// Mitsubishi GX Developer project: пресс 70 отключение при простое   PLC: Q04UDEH

PROGRAM MAIN
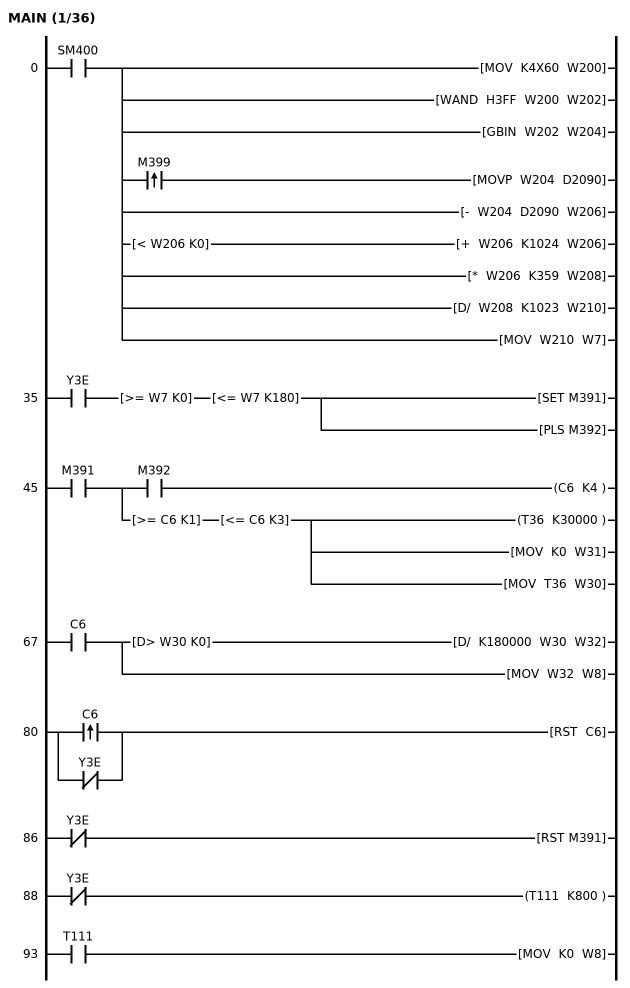
0     LD      SM400
      MOV     K4X60 W200
      WAND    H3FF W200 W202
      GBIN    W202 W204
      MPS
      ANDP    M399
      MOVP    W204 D2090
      MPP
      -       W204 D2090 W206
      MPS
      AND<    W206 K0
      +       W206 K1024 W206
      MPP
      *       W206 K359 W208
      D/      W208 K1023 W210
      MOV     W210 W7
35    LD      Y3E
      AND>=   W7 K0
      AND<=   W7 K180
      SET     M391
      PLS     M392
45    LD      M391
      MPS
      AND     M392
      OUT     C6 K4
      MPP
      AND>=   C6 K1
      AND<=   C6 K3
      OUTH    T36 K30000
      MOV     K0 W31
      MOV     T36 W30
67    LD      C6
      MPS
      ANDD>   W30 K0
      D/      K180000 W30 W32
      MPP
      MOV     W32 W8
80    LDP     C6
      ORI     Y3E
      RST     C6
86    LDI     Y3E
      RST     M391
88    LDI     Y3E
      OUT     T111 K800
93    LD      T111
      MOV     K0 W8
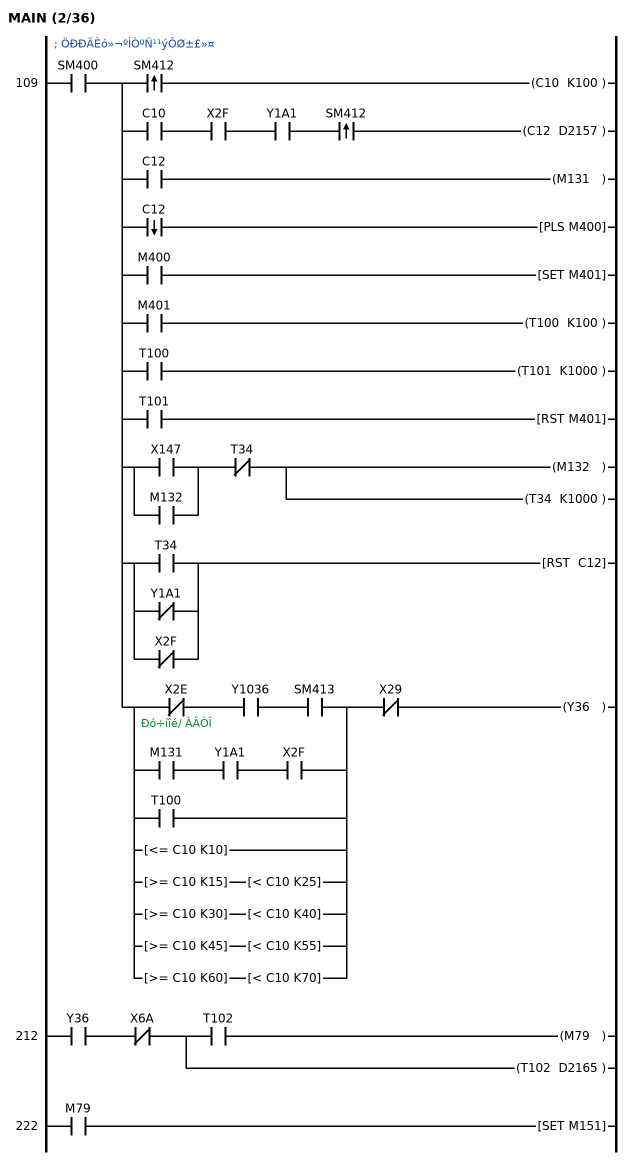
; 中心润滑和液压过载保护
109   LD      SM400
      MPS
      ANDP    SM412
      OUT     C10 K100
      MRD
      AND     C10
      AND     X2F
      AND     Y1A1
      ANDP    SM412
      OUT     C12 D2157
      MRD
      AND     C12
      OUT     M131
      MRD
      ANDF    C12
      PLS     M400
      MRD
      AND     M400
      SET     M401
      MRD
      AND     M401
      OUT     T100 K100
      MRD
      AND     T100
      OUT     T101 K1000
      MRD
      AND     T101
      RST     M401
      MRD
      LD      X147
      OR      M132
      ANB
      ANI     T34
      OUT     M132
      OUT     T34 K1000
      MRD
      LD      T34
      ORI     Y1A1
      ORI     X2F
      ANB
      RST     C12
      MPP
      LDI     X2E  ; Ручной/ АВТО
      AND     Y1036
      AND     SM413
      LD      M131
      AND     Y1A1
      AND     X2F
      ORB
      OR      T100
      OR<=    C10 K10
      LD>=    C10 K15
      AND<    C10 K25
      ORB
      LD>=    C10 K30
      AND<    C10 K40
      ORB
      LD>=    C10 K45
      AND<    C10 K55
      ORB
      LD>=    C10 K60
      AND<    C10 K70
      ORB
      ANB
      ANI     X29
      OUT     Y36
212   LD      Y36
      ANI     X6A
      MPS
      AND     T102
      OUT     M79
      MPP
      OUT     T102 D2165
222   LD      M79
      SET     M151
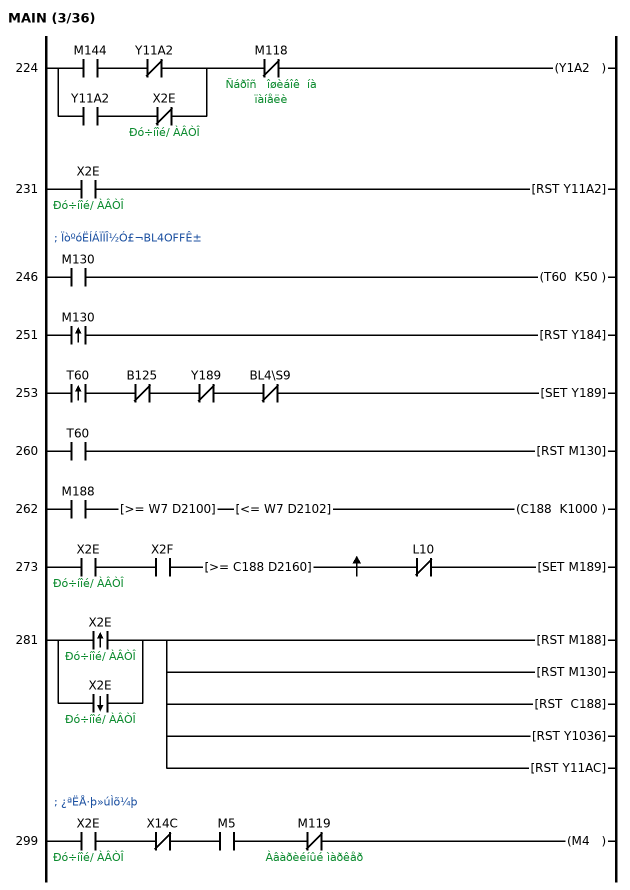
224   LD      M144
      ANI     Y11A2
      LD      Y11A2
      ANI     X2E  ; Ручной/ АВТО
      ORB
      ANI     M118  ; Сброс   ошибок  на панели
      OUT     Y1A2
231   LD      X2E  ; Ручной/ АВТО
      RST     Y11A2
; 向后送料衔接，BL4OFF时
246   LD      M130
      OUT     T60 K50
251   LDP     M130
      RST     Y184
253   LDP     T60
      ANI     B125
      ANI     Y189
      ANI     BL4\S9
      SET     Y189
260   LD      T60
      RST     M130
262   LD      M188
      AND>=   W7 D2100
      AND<=   W7 D2102
      OUT     C188 K1000
273   LD      X2E  ; Ручной/ АВТО
      AND     X2F
      AND>=   C188 D2160
      MEP
      ANI     L10
      SET     M189
281   LDP     X2E  ; Ручной/ АВТО
      ORF     X2E  ; Ручной/ АВТО
      RST     M188
      RST     M130
      RST     C188
      RST     Y1036
      RST     Y11AC
; 开伺服机条件
299   LD      X2E  ; Ручной/ АВТО
      ANI     X14C
      AND     M5
      ANI     M119  ; Аварийный маркер
      OUT     M4
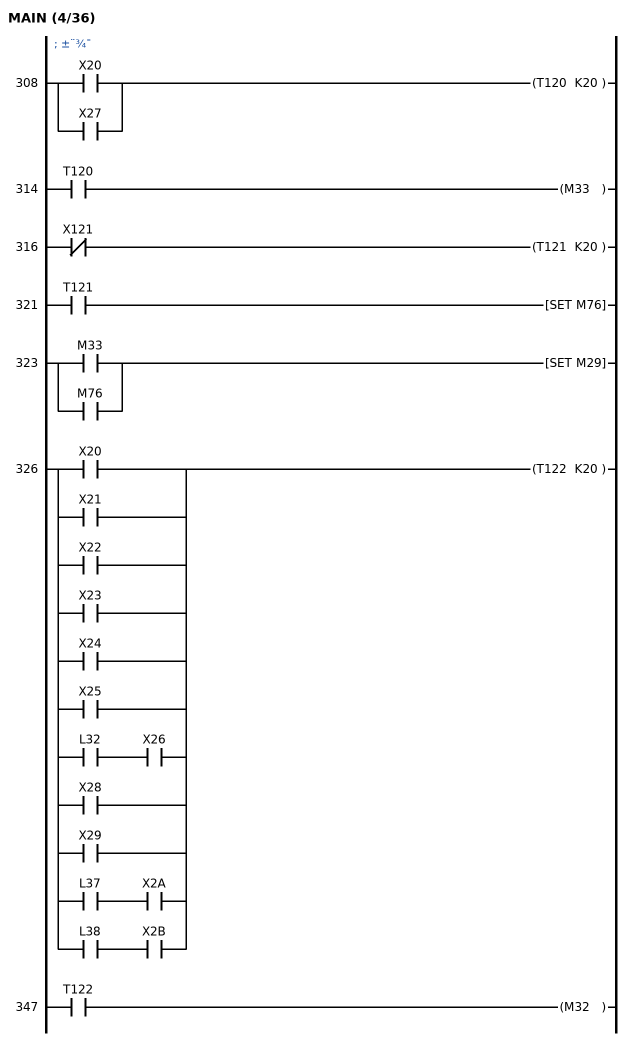
; ±¨¾¯
308   LD      X20
      OR      X27
      OUT     T120 K20
314   LD      T120
      OUT     M33
316   LDI     X121
      OUT     T121 K20
321   LD      T121
      SET     M76
323   LD      M33
      OR      M76
      SET     M29
326   LD      X20
      OR      X21
      OR      X22
      OR      X23
      OR      X24
      OR      X25
      LD      L32
      AND     X26
      ORB
      OR      X28
      OR      X29
      LD      L37
      AND     X2A
      ORB
      LD      L38
      AND     X2B
      ORB
      OUT     T122 K20
347   LD      T122
      OUT     M32
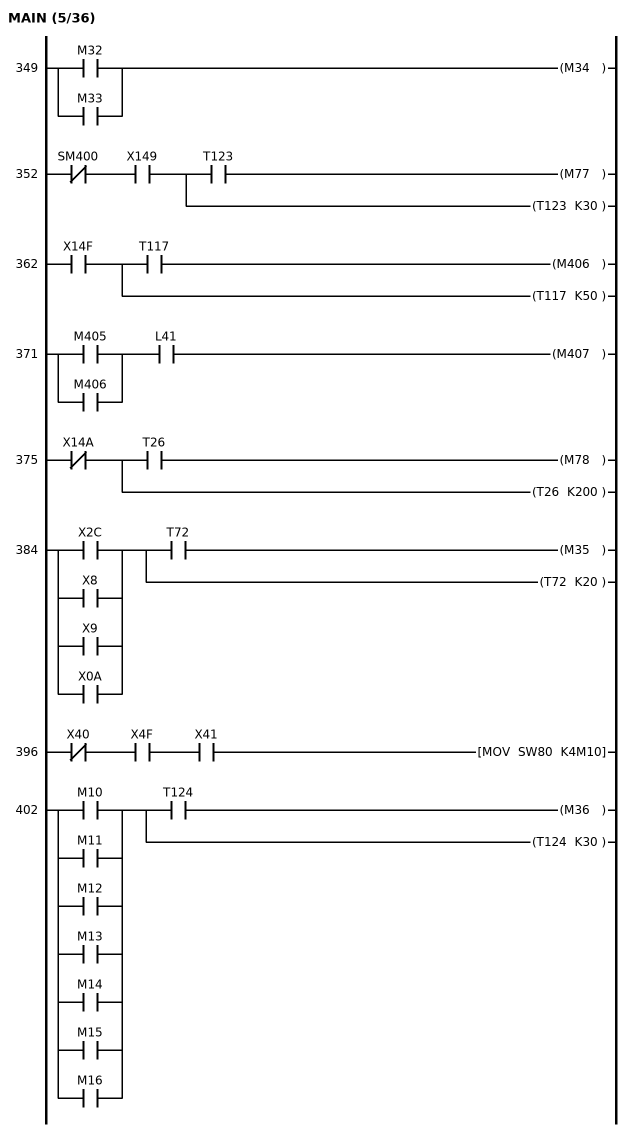
349   LD      M32
      OR      M33
      OUT     M34
352   LDI     SM400
      AND     X149
      MPS
      AND     T123
      OUT     M77
      MPP
      OUT     T123 K30
362   LD      X14F
      MPS
      AND     T117
      OUT     M406
      MPP
      OUT     T117 K50
371   LD      M405
      OR      M406
      AND     L41
      OUT     M407
375   LDI     X14A
      MPS
      AND     T26
      OUT     M78
      MPP
      OUT     T26 K200
384   LD      X2C
      OR      X8
      OR      X9
      OR      X0A
      MPS
      AND     T72
      OUT     M35
      MPP
      OUT     T72 K20
396   LDI     X40
      AND     X4F
      AND     X41
      MOV     SW80 K4M10
402   LD      M10
      OR      M11
      OR      M12
      OR      M13
      OR      M14
      OR      M15
      OR      M16
      MPS
      AND     T124
      OUT     M36
      MPP
      OUT     T124 K30
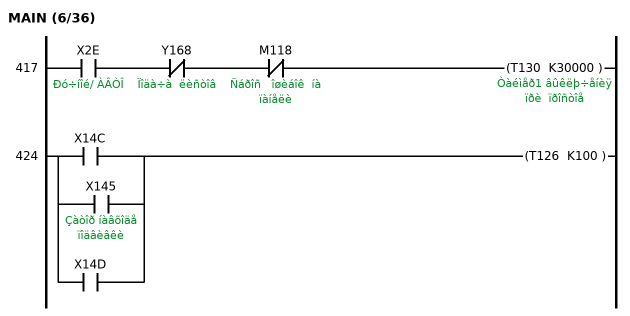
417   LD      X2E  ; Ручной/ АВТО
      ANI     Y168  ; Подача  листов
      ANI     M118  ; Сброс   ошибок  на панели
      OUT     T130 K30000  ; Таймер1 выключения при  простое
424   LD      X14C
      OR      X145  ; Затор навходе   подвивки
      OR      X14D
      OUTH    T126 K100
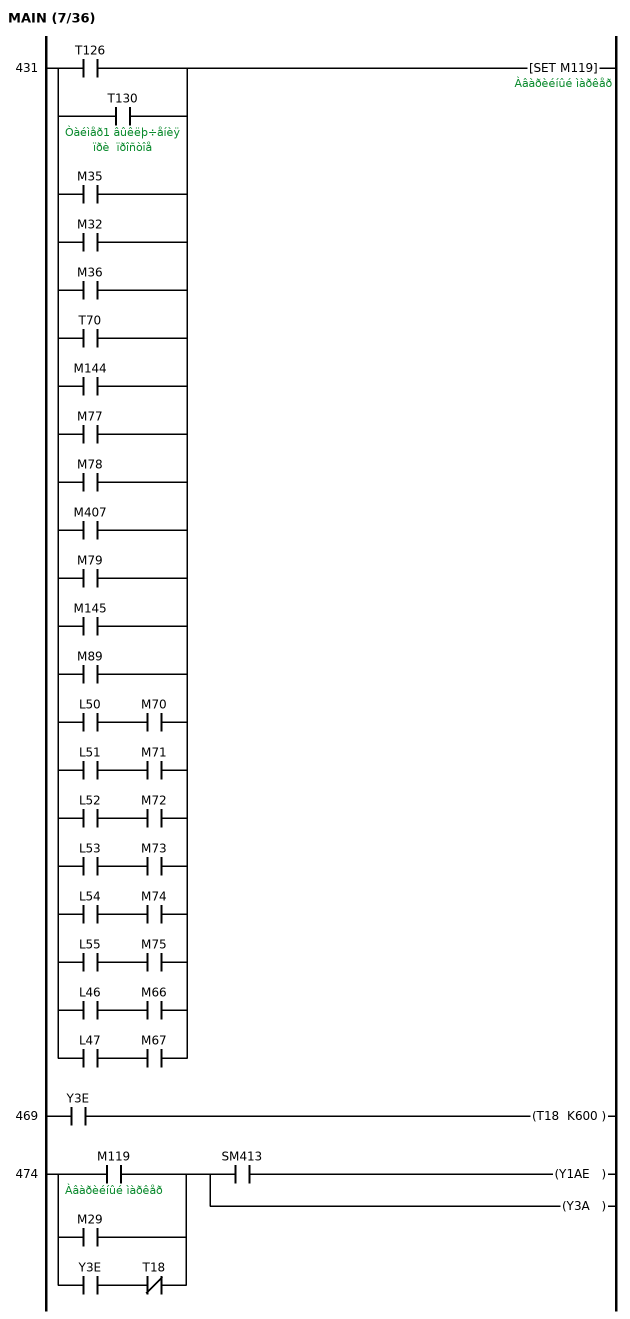
431   LD      T126
      OR      T130  ; Таймер1 выключения при  простое
      OR      M35
      OR      M32
      OR      M36
      OR      T70
      OR      M144
      OR      M77
      OR      M78
      OR      M407
      OR      M79
      OR      M145
      OR      M89
      LD      L50
      AND     M70
      ORB
      LD      L51
      AND     M71
      ORB
      LD      L52
      AND     M72
      ORB
      LD      L53
      AND     M73
      ORB
      LD      L54
      AND     M74
      ORB
      LD      L55
      AND     M75
      ORB
      LD      L46
      AND     M66
      ORB
      LD      L47
      AND     M67
      ORB
      SET     M119  ; Аварийный маркер
469   LD      Y3E
      OUT     T18 K600
474   LD      M119  ; Аварийный маркер
      OR      M29
      LD      Y3E
      ANI     T18
      ORB
      MPS
      AND     SM413
      OUT     Y1AE
      MPP
      OUT     Y3A
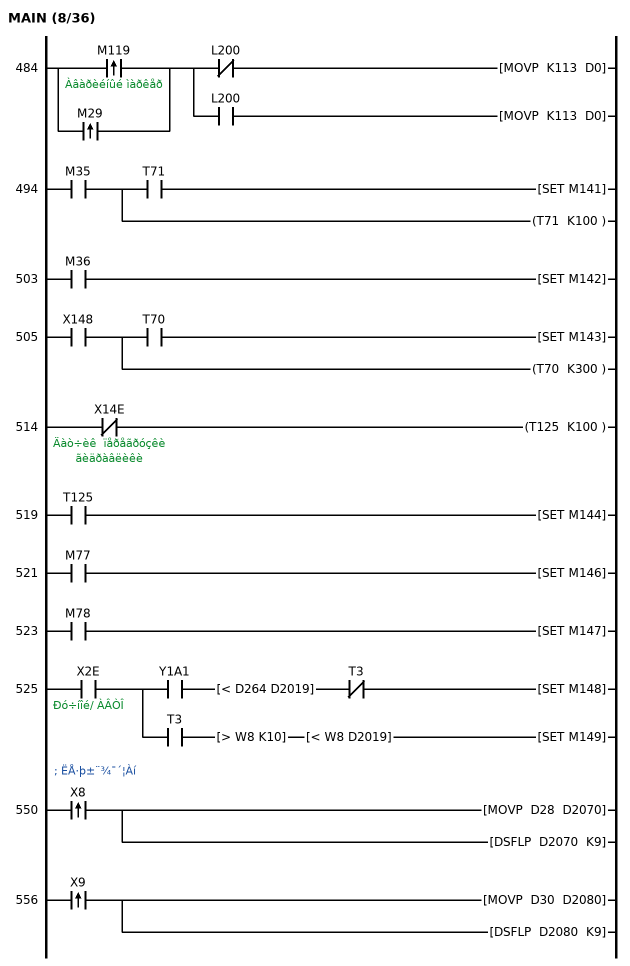
484   LDP     M119  ; Аварийный маркер
      ORP     M29
      MPS
      ANI     L200
      MOVP    K113 D0
      MPP
      AND     L200
      MOVP    K113 D0
494   LD      M35
      MPS
      AND     T71
      SET     M141
      MPP
      OUT     T71 K100
503   LD      M36
      SET     M142
505   LD      X148
      MPS
      AND     T70
      SET     M143
      MPP
      OUT     T70 K300
514   LDI     X14E  ; Датчик  перегрузки гидравлики
      OUTH    T125 K100
519   LD      T125
      SET     M144
521   LD      M77
      SET     M146
523   LD      M78
      SET     M147
525   LD      X2E  ; Ручной/ АВТО
      MPS
      AND     Y1A1
      AND<    D264 D2019
      ANI     T3
      SET     M148
      MPP
      AND     T3
      AND>    W8 K10
      AND<    W8 D2019
      SET     M149
; 伺服报警处理
550   LDP     X8
      MOVP    D28 D2070
      DSFLP   D2070 K9
556   LDP     X9
      MOVP    D30 D2080
      DSFLP   D2080 K9
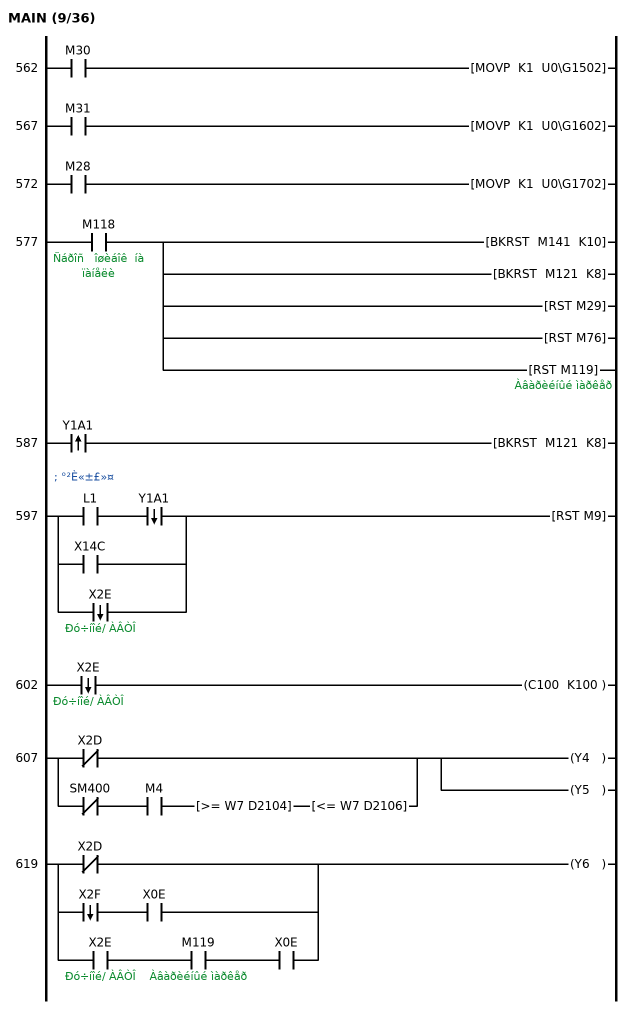
562   LD      M30
      MOVP    K1 U0\G1502
567   LD      M31
      MOVP    K1 U0\G1602
572   LD      M28
      MOVP    K1 U0\G1702
577   LD      M118  ; Сброс   ошибок  на панели
      BKRST   M141 K10
      BKRST   M121 K8
      RST     M29
      RST     M76
      RST     M119  ; Аварийный маркер
587   LDP     Y1A1
      BKRST   M121 K8
; 安全保护
597   LD      L1
      ANDF    Y1A1
      OR      X14C
      ORF     X2E  ; Ручной/ АВТО
      RST     M9
602   LDF     X2E  ; Ручной/ АВТО
      OUT     C100 K100
607   LDI     X2D
      LDI     SM400
      AND     M4
      AND>=   W7 D2104
      AND<=   W7 D2106
      ORB
      OUT     Y4
      OUT     Y5
619   LDI     X2D
      LDF     X2F
      AND     X0E
      ORB
      LD      X2E  ; Ручной/ АВТО
      AND     M119  ; Аварийный маркер
      AND     X0E
      ORB
      OUT     Y6
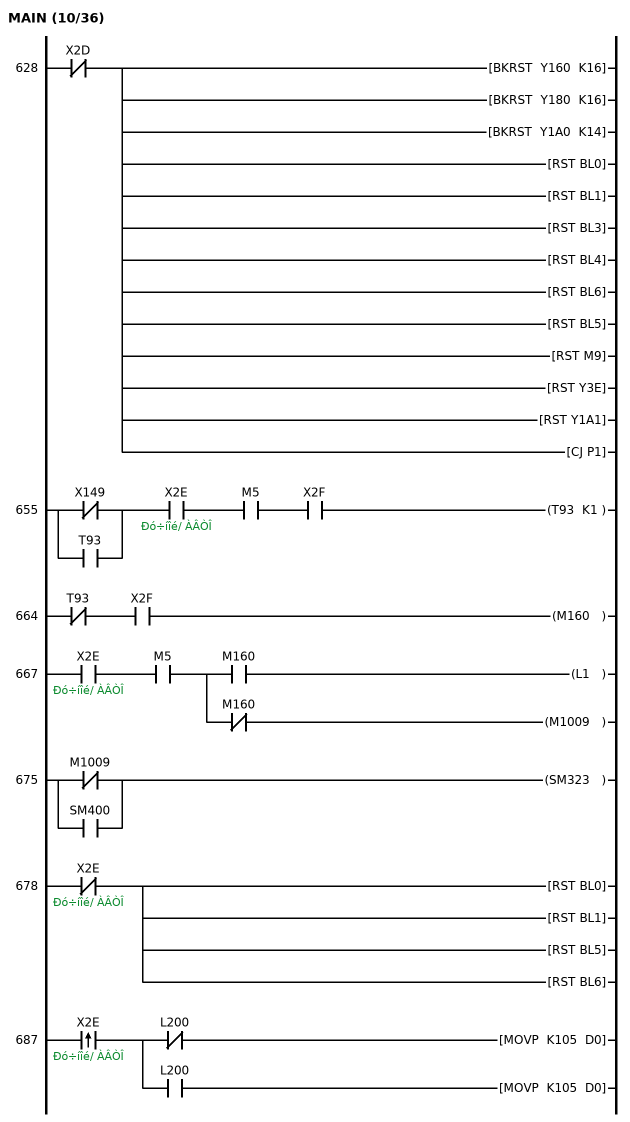
628   LDI     X2D
      BKRST   Y160 K16
      BKRST   Y180 K16
      BKRST   Y1A0 K14
      RST     BL0
      RST     BL1
      RST     BL3
      RST     BL4
      RST     BL6
      RST     BL5
      RST     M9
      RST     Y3E
      RST     Y1A1
      CJ      P1
655   LDI     X149
      OR      T93
      AND     X2E  ; Ручной/ АВТО
      AND     M5
      AND     X2F
      OUT     T93 K1
664   LDI     T93
      AND     X2F
      OUT     M160
667   LD      X2E  ; Ручной/ АВТО
      AND     M5
      MPS
      AND     M160
      OUT     L1
      MPP
      ANI     M160
      OUT     M1009
675   LDI     M1009
      OR      SM400
      OUT     SM323
678   LDI     X2E  ; Ручной/ АВТО
      RST     BL0
      RST     BL1
      RST     BL5
      RST     BL6
687   LDP     X2E  ; Ручной/ АВТО
      MPS
      ANI     L200
      MOVP    K105 D0
      MPP
      AND     L200
      MOVP    K105 D0
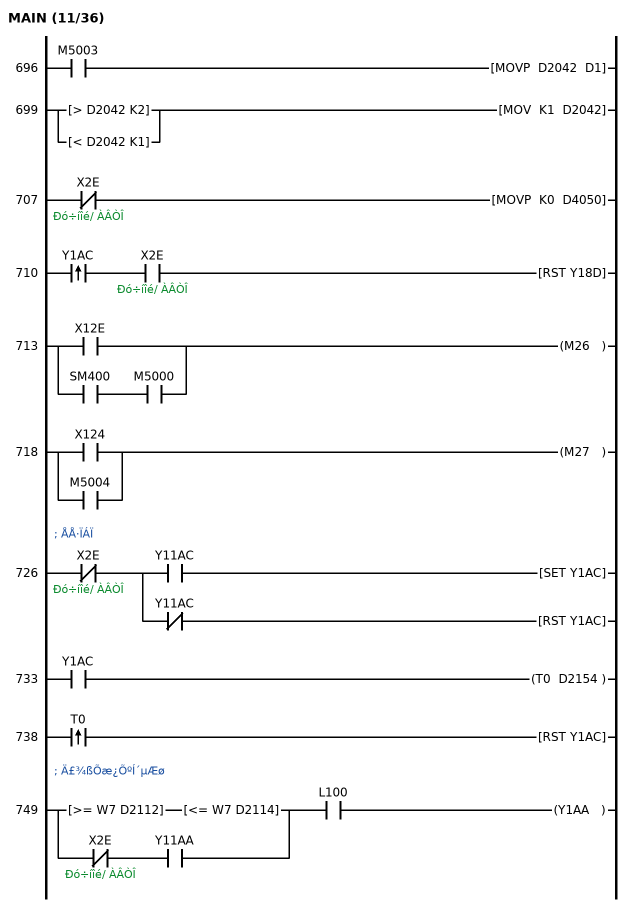
696   LD      M5003
      MOVP    D2042 D1
699   LD>     D2042 K2
      OR<     D2042 K1
      MOV     K1 D2042
707   LDI     X2E  ; Ручной/ АВТО
      MOVP    K0 D4050
710   LDP     Y1AC
      AND     X2E  ; Ручной/ АВТО
      RST     Y18D
713   LD      X12E
      LD      SM400
      AND     M5000
      ORB
      OUT     M26
718   LD      X124
      OR      M5004
      OUT     M27
; ÅÅ·ÏÁÏ
726   LDI     X2E  ; Ручной/ АВТО
      MPS
      AND     Y11AC
      SET     Y1AC
      MPP
      ANI     Y11AC
      RST     Y1AC
733   LD      Y1AC
      OUTH    T0 D2154
738   LDP     T0
      RST     Y1AC
; Ä£¾ßÕæ¿ÕºÍ´µÆø
749   LD>=    W7 D2112
      AND<=   W7 D2114
      LDI     X2E  ; Ручной/ АВТО
      AND     Y11AA
      ORB
      AND     L100
      OUT     Y1AA
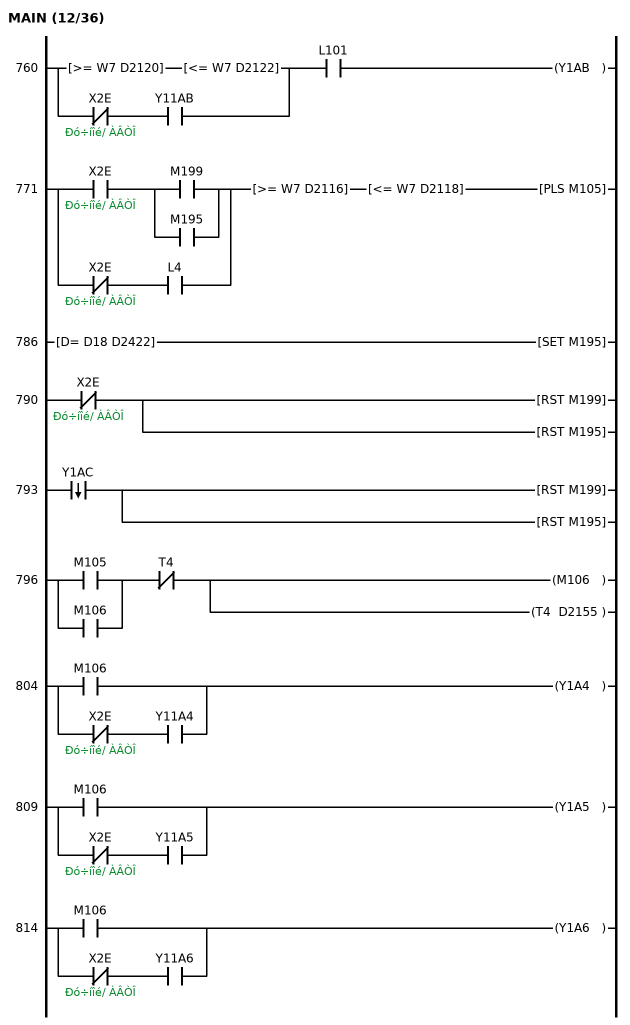
760   LD>=    W7 D2120
      AND<=   W7 D2122
      LDI     X2E  ; Ручной/ АВТО
      AND     Y11AB
      ORB
      AND     L101
      OUT     Y1AB
771   LD      X2E  ; Ручной/ АВТО
      LD      M199
      OR      M195
      ANB
      LDI     X2E  ; Ручной/ АВТО
      AND     L4
      ORB
      AND>=   W7 D2116
      AND<=   W7 D2118
      PLS     M105
786   LDD=    D18 D2422
      SET     M195
790   LDI     X2E  ; Ручной/ АВТО
      RST     M199
      RST     M195
793   LDF     Y1AC
      RST     M199
      RST     M195
796   LD      M105
      OR      M106
      ANI     T4
      OUT     M106
      OUTH    T4 D2155
804   LD      M106
      LDI     X2E  ; Ручной/ АВТО
      AND     Y11A4
      ORB
      OUT     Y1A4
809   LD      M106
      LDI     X2E  ; Ручной/ АВТО
      AND     Y11A5
      ORB
      OUT     Y1A5
814   LD      M106
      LDI     X2E  ; Ручной/ АВТО
      AND     Y11A6
      ORB
      OUT     Y1A6
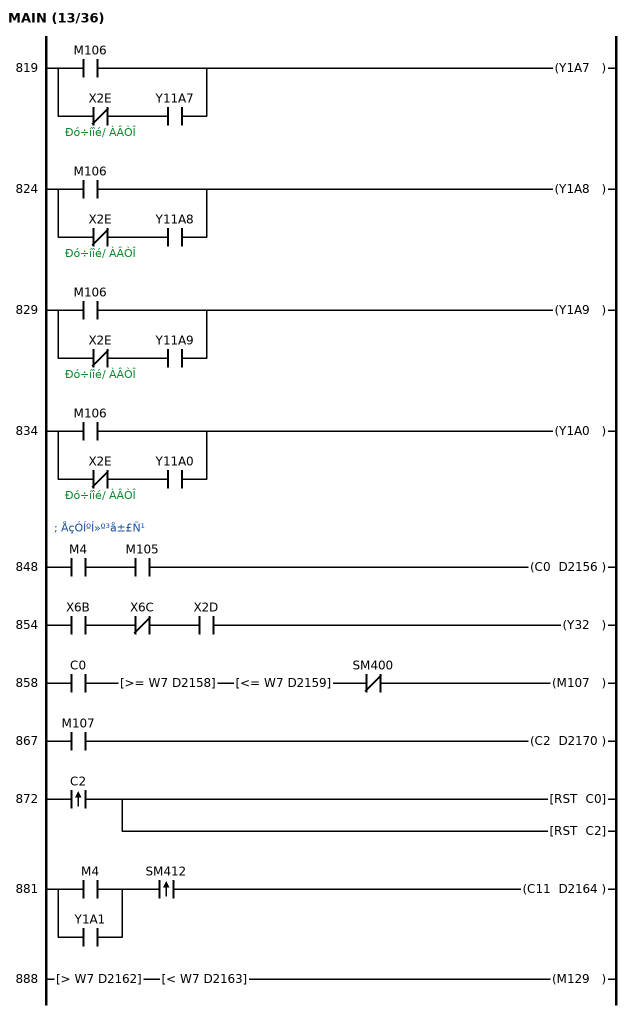
819   LD      M106
      LDI     X2E  ; Ручной/ АВТО
      AND     Y11A7
      ORB
      OUT     Y1A7
824   LD      M106
      LDI     X2E  ; Ручной/ АВТО
      AND     Y11A8
      ORB
      OUT     Y1A8
829   LD      M106
      LDI     X2E  ; Ручной/ АВТО
      AND     Y11A9
      ORB
      OUT     Y1A9
834   LD      M106
      LDI     X2E  ; Ручной/ АВТО
      AND     Y11A0
      ORB
      OUT     Y1A0
; ÅçÓÍºÍ»º³å±£Ñ¹
848   LD      M4
      AND     M105
      OUT     C0 D2156
854   LD      X6B
      ANI     X6C
      AND     X2D
      OUT     Y32
858   LD      C0
      AND>=   W7 D2158
      AND<=   W7 D2159
      ANI     SM400
      OUT     M107
867   LD      M107
      OUT     C2 D2170
872   LDP     C2
      RST     C0
      RST     C2
881   LD      M4
      OR      Y1A1
      ANDP    SM412
      OUT     C11 D2164
888   LD>     W7 D2162
      AND<    W7 D2163
      OUT     M129
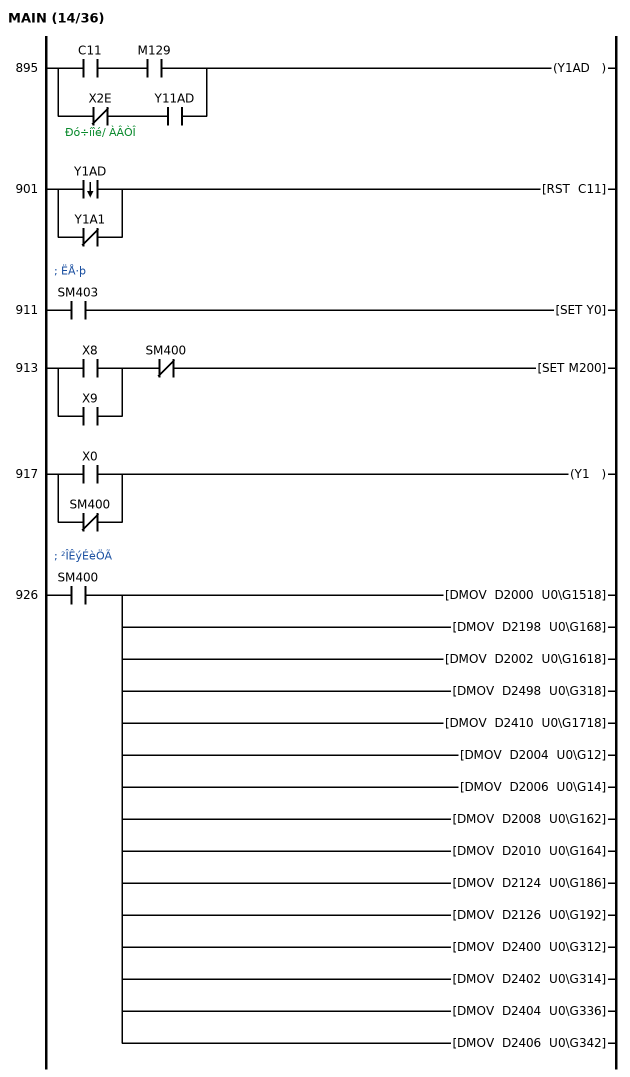
895   LD      C11
      AND     M129
      LDI     X2E  ; Ручной/ АВТО
      AND     Y11AD
      ORB
      OUT     Y1AD
901   LDF     Y1AD
      ORI     Y1A1
      RST     C11
; ËÅ·þ
911   LD      SM403
      SET     Y0
913   LD      X8
      OR      X9
      ANI     SM400
      SET     M200
917   LD      X0
      ORI     SM400
      OUT     Y1
; 参数设置
926   LD      SM400
      DMOV    D2000 U0\G1518
      DMOV    D2198 U0\G168
      DMOV    D2002 U0\G1618
      DMOV    D2498 U0\G318
      DMOV    D2410 U0\G1718
      DMOV    D2004 U0\G12
      DMOV    D2006 U0\G14
      DMOV    D2008 U0\G162
      DMOV    D2010 U0\G164
      DMOV    D2124 U0\G186
      DMOV    D2126 U0\G192
      DMOV    D2400 U0\G312
      DMOV    D2402 U0\G314
      DMOV    D2404 U0\G336
      DMOV    D2406 U0\G342
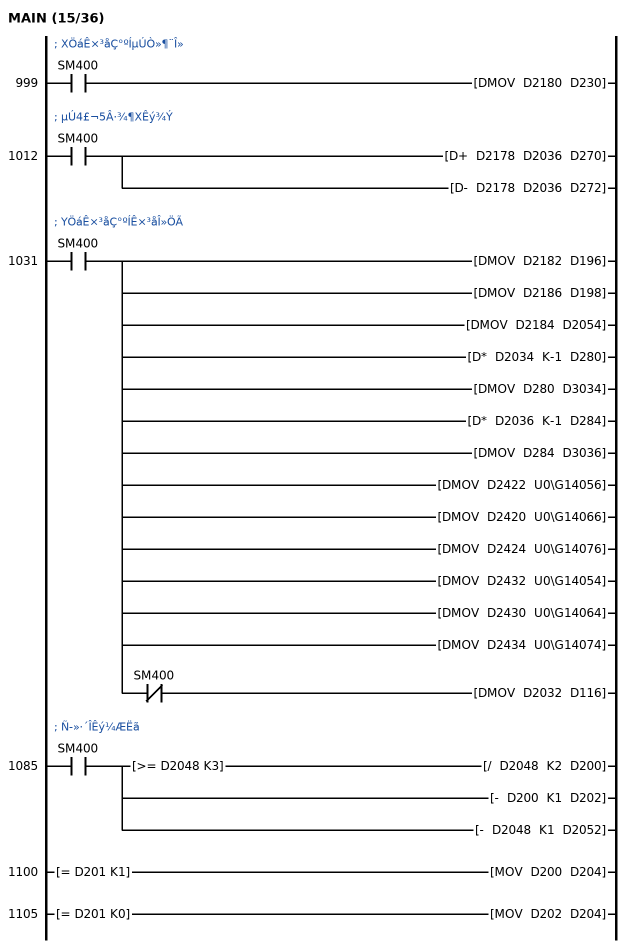
; X轴首冲前和第一定位
999   LD      SM400
      DMOV    D2180 D230
; 第4，5路径X数据
1012  LD      SM400
      D+      D2178 D2036 D270
      D-      D2178 D2036 D272
; Y轴首冲前和首冲位置
1031  LD      SM400
      DMOV    D2182 D196
      DMOV    D2186 D198
      DMOV    D2184 D2054
      D*      D2034 K-1 D280
      DMOV    D280 D3034
      D*      D2036 K-1 D284
      DMOV    D284 D3036
      DMOV    D2422 U0\G14056
      DMOV    D2420 U0\G14066
      DMOV    D2424 U0\G14076
      DMOV    D2432 U0\G14054
      DMOV    D2430 U0\G14064
      DMOV    D2434 U0\G14074
      ANI     SM400
      DMOV    D2032 D116
; 循环次数计算
1085  LD      SM400
      MPS
      AND>=   D2048 K3
      /       D2048 K2 D200
      MPP
      -       D200 K1 D202
      -       D2048 K1 D2052
1100  LD=     D201 K1
      MOV     D200 D204
1105  LD=     D201 K0
      MOV     D202 D204
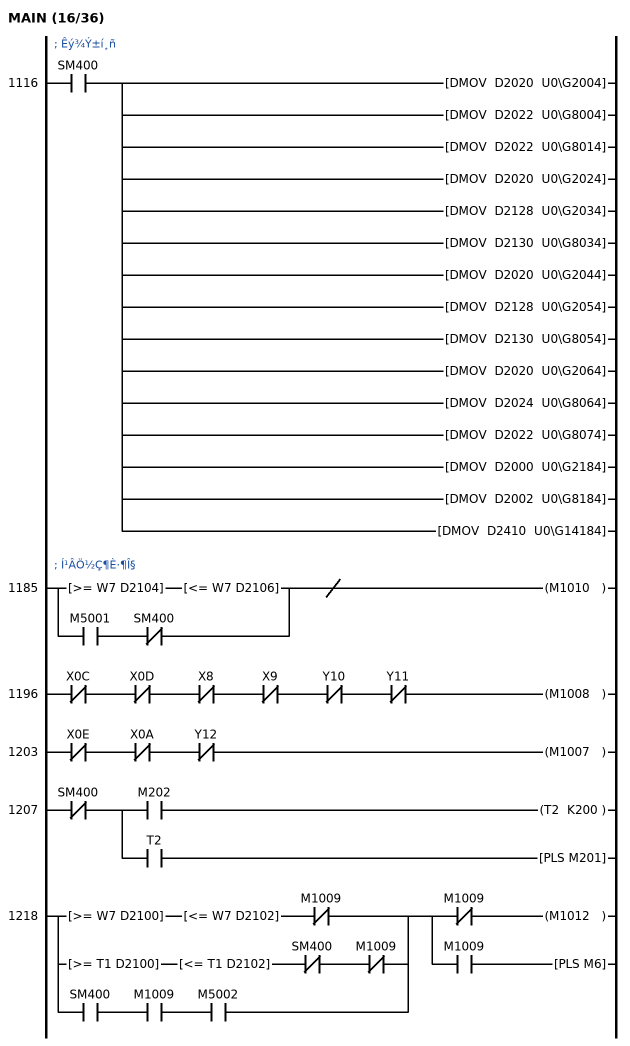
; 数据表格
1116  LD      SM400
      DMOV    D2020 U0\G2004
      DMOV    D2022 U0\G8004
      DMOV    D2022 U0\G8014
      DMOV    D2020 U0\G2024
      DMOV    D2128 U0\G2034
      DMOV    D2130 U0\G8034
      DMOV    D2020 U0\G2044
      DMOV    D2128 U0\G2054
      DMOV    D2130 U0\G8054
      DMOV    D2020 U0\G2064
      DMOV    D2024 U0\G8064
      DMOV    D2022 U0\G8074
      DMOV    D2000 U0\G2184
      DMOV    D2002 U0\G8184
      DMOV    D2410 U0\G14184
; 凸轮角度范围
1185  LD>=    W7 D2104
      AND<=   W7 D2106
      LD      M5001
      ANI     SM400
      ORB
      INV
      OUT     M1010
1196  LDI     X0C
      ANI     X0D
      ANI     X8
      ANI     X9
      ANI     Y10
      ANI     Y11
      OUT     M1008
1203  LDI     X0E
      ANI     X0A
      ANI     Y12
      OUT     M1007
1207  LDI     SM400
      MPS
      AND     M202
      OUT     T2 K200
      MPP
      AND     T2
      PLS     M201
1218  LD>=    W7 D2100
      AND<=   W7 D2102
      ANI     M1009
      LD>=    T1 D2100
      AND<=   T1 D2102
      ANI     SM400
      ANI     M1009
      ORB
      LD      SM400
      AND     M1009
      AND     M5002
      ORB
      MPS
      ANI     M1009
      OUT     M1012
      MPP
      AND     M1009
      PLS     M6
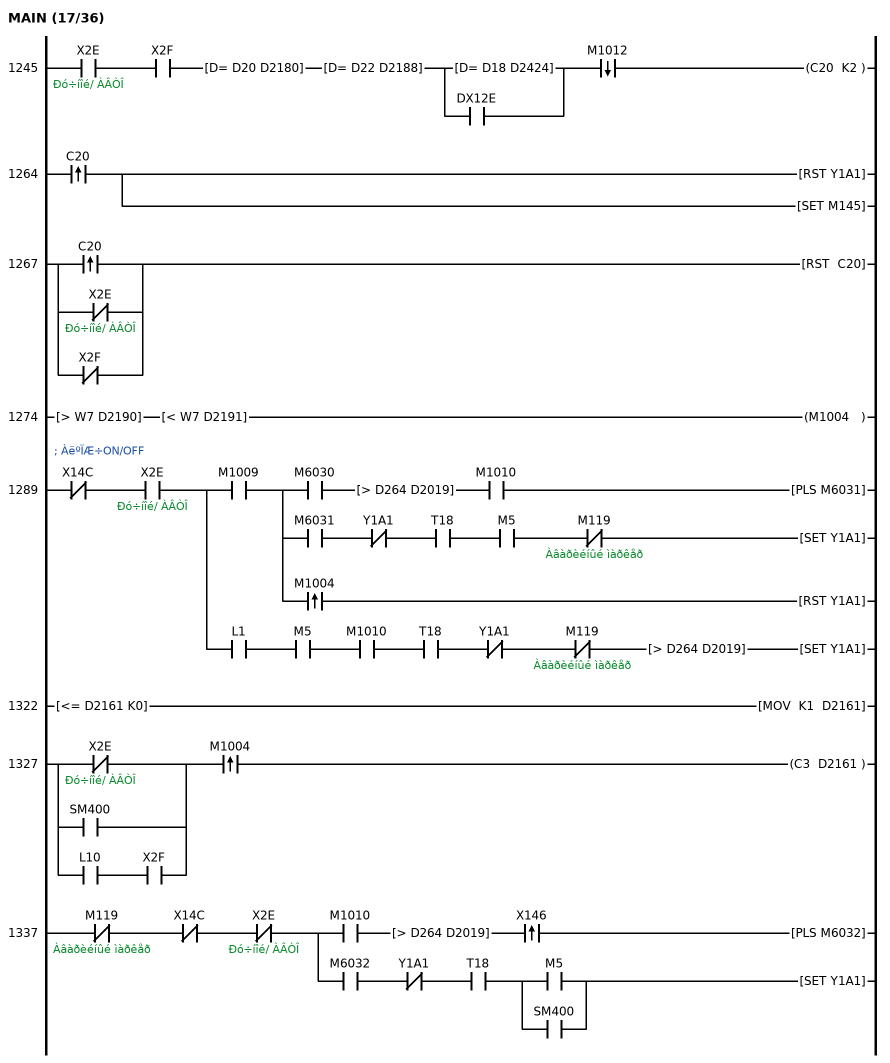
1245  LD      X2E  ; Ручной/ АВТО
      AND     X2F
      ANDD=   D20 D2180
      ANDD=   D22 D2188
      LDD=    D18 D2424
      OR      DX12E
      ANB
      ANDF    M1012
      OUT     C20 K2
1264  LDP     C20
      RST     Y1A1
      SET     M145
1267  LDP     C20
      ORI     X2E  ; Ручной/ АВТО
      ORI     X2F
      RST     C20
1274  LD>     W7 D2190
      AND<    W7 D2191
      OUT     M1004
; 离合器ON/OFF
1289  LDI     X14C
      AND     X2E  ; Ручной/ АВТО
      MPS
      AND     M1009
      MPS
      AND     M6030
      AND>    D264 D2019
      AND     M1010
      PLS     M6031
      MRD
      AND     M6031
      ANI     Y1A1
      AND     T18
      AND     M5
      ANI     M119  ; Аварийный маркер
      SET     Y1A1
      MPP
      ANDP    M1004
      RST     Y1A1
      MPP
      AND     L1
      AND     M5
      AND     M1010
      AND     T18
      ANI     Y1A1
      ANI     M119  ; Аварийный маркер
      AND>    D264 D2019
      SET     Y1A1
1322  LD<=    D2161 K0
      MOV     K1 D2161
1327  LDI     X2E  ; Ручной/ АВТО
      OR      SM400
      LD      L10
      AND     X2F
      ORB
      ANDP    M1004
      OUT     C3 D2161
1337  LDI     M119  ; Аварийный маркер
      ANI     X14C
      ANI     X2E  ; Ручной/ АВТО
      MPS
      AND     M1010
      AND>    D264 D2019
      ANDP    X146
      PLS     M6032
      MPP
      AND     M6032
      ANI     Y1A1
      AND     T18
      LD      M5
      OR      SM400
      ANB
      SET     Y1A1
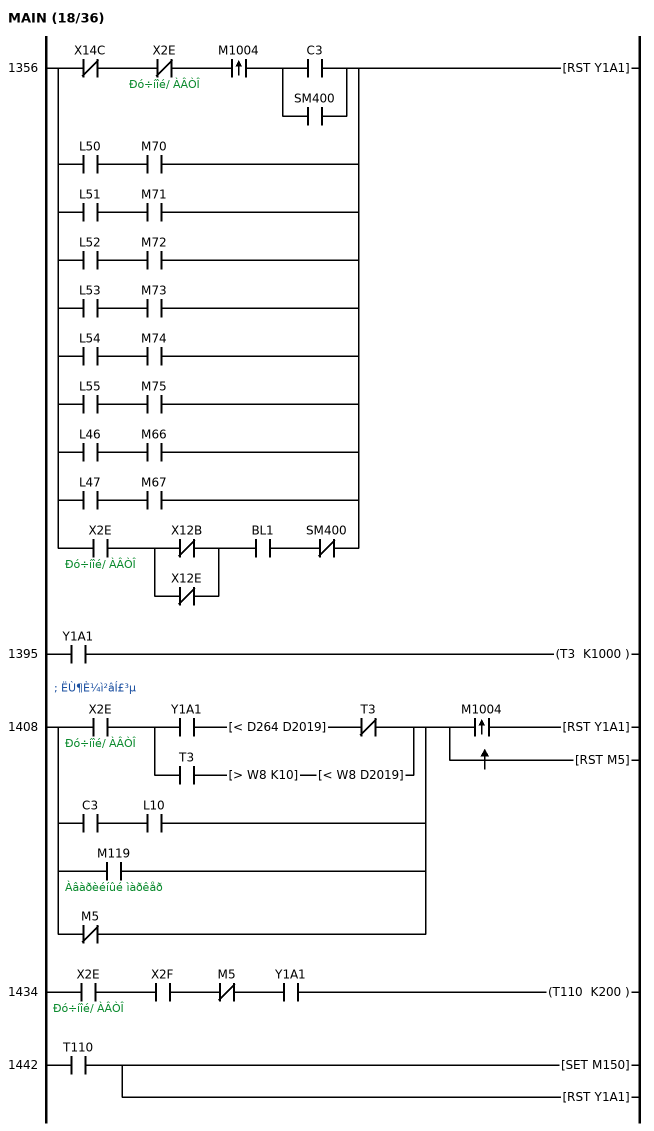
1356  LDI     X14C
      ANI     X2E  ; Ручной/ АВТО
      ANDP    M1004
      LD      C3
      OR      SM400
      ANB
      LD      L50
      AND     M70
      ORB
      LD      L51
      AND     M71
      ORB
      LD      L52
      AND     M72
      ORB
      LD      L53
      AND     M73
      ORB
      LD      L54
      AND     M74
      ORB
      LD      L55
      AND     M75
      ORB
      LD      L46
      AND     M66
      ORB
      LD      L47
      AND     M67
      ORB
      LD      X2E  ; Ручной/ АВТО
      LDI     X12B
      ORI     X12E
      ANB
      AND     BL1
      ANI     SM400
      ORB
      RST     Y1A1
1395  LD      Y1A1
      OUT     T3 K1000
; 速度检测停车
1408  LD      X2E  ; Ручной/ АВТО
      LD      Y1A1
      AND<    D264 D2019
      ANI     T3
      LD      T3
      AND>    W8 K10
      AND<    W8 D2019
      ORB
      ANB
      LD      C3
      AND     L10
      ORB
      OR      M119  ; Аварийный маркер
      ORI     M5
      MPS
      ANDP    M1004
      RST     Y1A1
      MPP
      MEP
      RST     M5
1434  LD      X2E  ; Ручной/ АВТО
      AND     X2F
      ANI     M5
      AND     Y1A1
      OUT     T110 K200
1442  LD      T110
      SET     M150
      RST     Y1A1
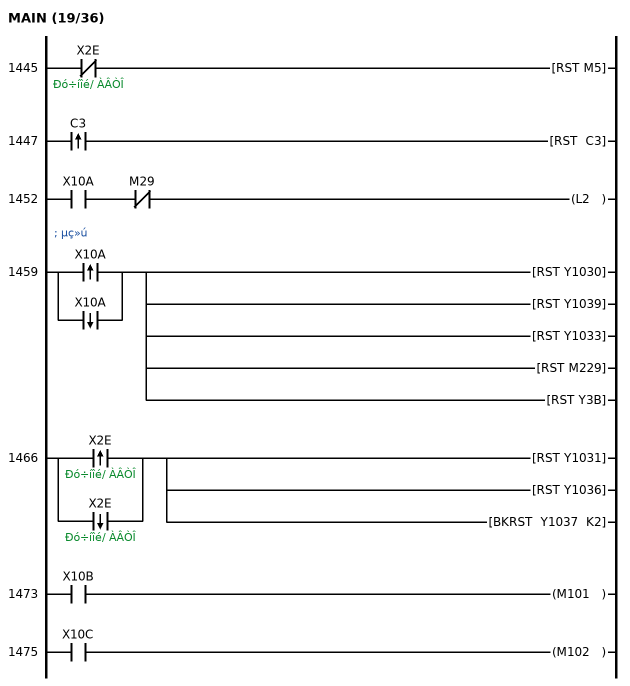
1445  LDI     X2E  ; Ручной/ АВТО
      RST     M5
1447  LDP     C3
      RST     C3
1452  LD      X10A
      ANI     M29
      OUT     L2
; µç»ú
1459  LDP     X10A
      ORF     X10A
      RST     Y1030
      RST     Y1039
      RST     Y1033
      RST     M229
      RST     Y3B
1466  LDP     X2E  ; Ручной/ АВТО
      ORF     X2E  ; Ручной/ АВТО
      RST     Y1031
      RST     Y1036
      BKRST   Y1037 K2
1473  LD      X10B
      OUT     M101
1475  LD      X10C
      OUT     M102
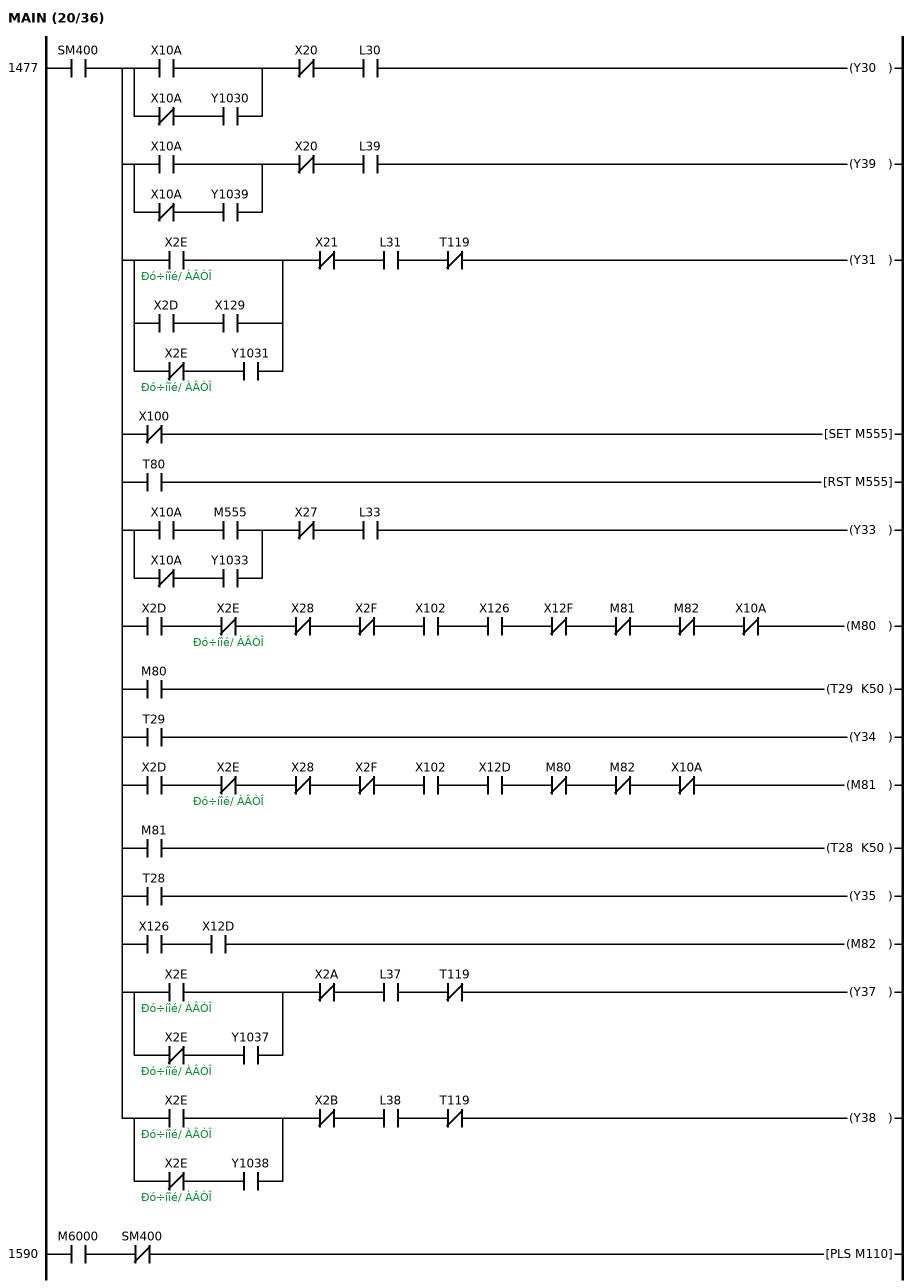
1477  LD      SM400
      MPS
      LD      X10A
      LDI     X10A
      AND     Y1030
      ORB
      ANB
      ANI     X20
      AND     L30
      OUT     Y30
      MRD
      LD      X10A
      LDI     X10A
      AND     Y1039
      ORB
      ANB
      ANI     X20
      AND     L39
      OUT     Y39
      MRD
      LD      X2E  ; Ручной/ АВТО
      LD      X2D
      AND     X129
      ORB
      LDI     X2E  ; Ручной/ АВТО
      AND     Y1031
      ORB
      ANB
      ANI     X21
      AND     L31
      ANI     T119
      OUT     Y31
      MRD
      ANI     X100
      SET     M555
      MRD
      AND     T80
      RST     M555
      MRD
      LD      X10A
      AND     M555
      LDI     X10A
      AND     Y1033
      ORB
      ANB
      ANI     X27
      AND     L33
      OUT     Y33
      MRD
      AND     X2D
      ANI     X2E  ; Ручной/ АВТО
      ANI     X28
      ANI     X2F
      AND     X102
      AND     X126
      ANI     X12F
      ANI     M81
      ANI     M82
      ANI     X10A
      OUT     M80
      MRD
      AND     M80
      OUT     T29 K50
      MRD
      AND     T29
      OUT     Y34
      MRD
      AND     X2D
      ANI     X2E  ; Ручной/ АВТО
      ANI     X28
      ANI     X2F
      AND     X102
      AND     X12D
      ANI     M80
      ANI     M82
      ANI     X10A
      OUT     M81
      MRD
      AND     M81
      OUT     T28 K50
      MRD
      AND     T28
      OUT     Y35
      MRD
      AND     X126
      AND     X12D
      OUT     M82
      MRD
      LD      X2E  ; Ручной/ АВТО
      LDI     X2E  ; Ручной/ АВТО
      AND     Y1037
      ORB
      ANB
      ANI     X2A
      AND     L37
      ANI     T119
      OUT     Y37
      MPP
      LD      X2E  ; Ручной/ АВТО
      LDI     X2E  ; Ручной/ АВТО
      AND     Y1038
      ORB
      ANB
      ANI     X2B
      AND     L38
      ANI     T119
      OUT     Y38
1590  LD      M6000
      ANI     SM400
      PLS     M110
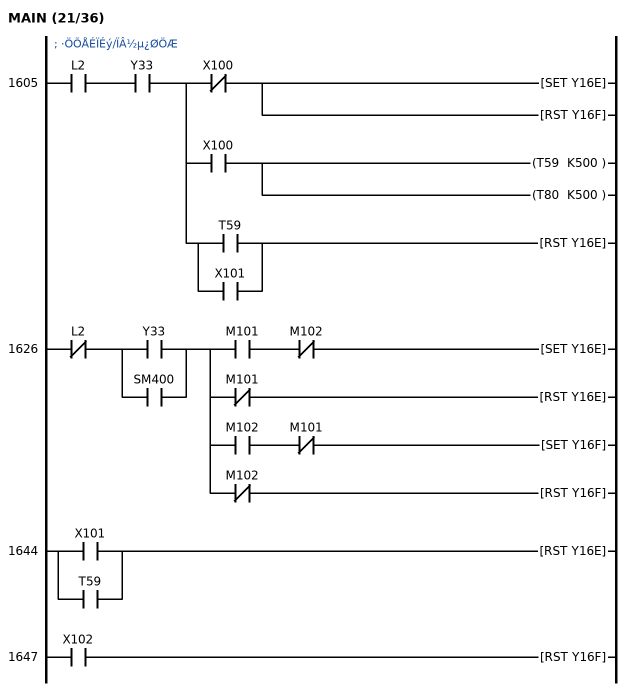
; 分张上升/下降控制
1605  LD      L2
      AND     Y33
      MPS
      ANI     X100
      SET     Y16E
      RST     Y16F
      MRD
      AND     X100
      OUTH    T59 K500
      OUT     T80 K500
      MPP
      LD      T59
      OR      X101
      ANB
      RST     Y16E
1626  LDI     L2
      LD      Y33
      OR      SM400
      ANB
      MPS
      AND     M101
      ANI     M102
      SET     Y16E
      MRD
      ANI     M101
      RST     Y16E
      MRD
      AND     M102
      ANI     M101
      SET     Y16F
      MPP
      ANI     M102
      RST     Y16F
1644  LD      X101
      OR      T59
      RST     Y16E
1647  LD      X102
      RST     Y16F
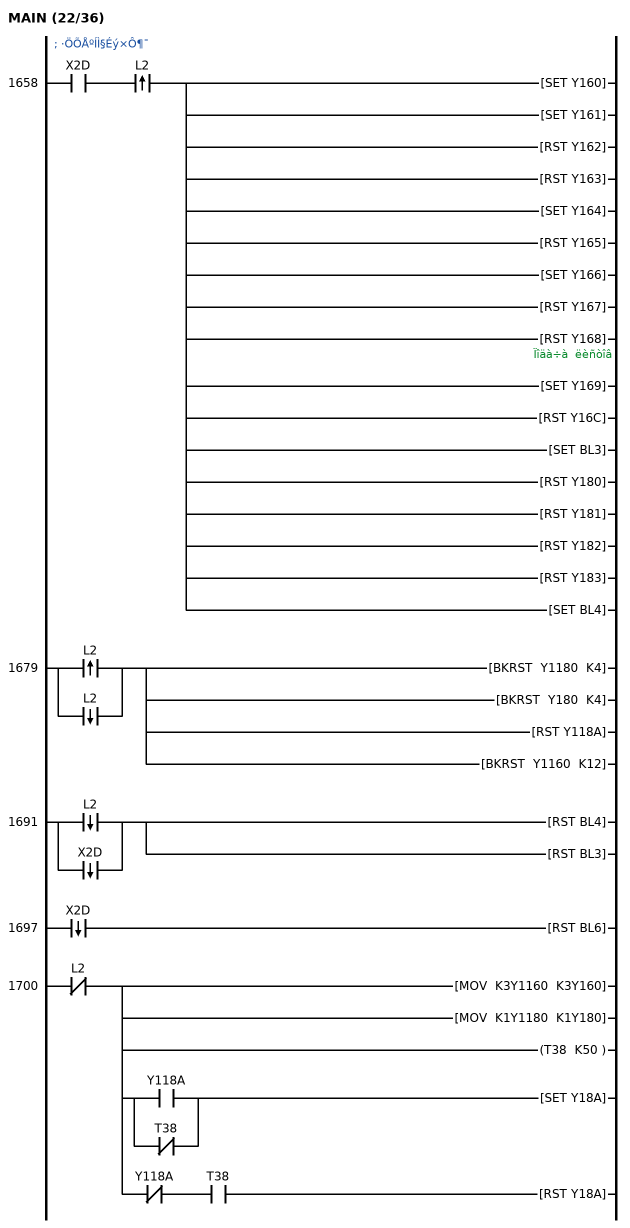
; 分张和抬升自动
1658  LD      X2D
      ANDP    L2
      SET     Y160
      SET     Y161
      RST     Y162
      RST     Y163
      SET     Y164
      RST     Y165
      SET     Y166
      RST     Y167
      RST     Y168  ; Подача  листов
      SET     Y169
      RST     Y16C
      SET     BL3
      RST     Y180
      RST     Y181
      RST     Y182
      RST     Y183
      SET     BL4
1679  LDP     L2
      ORF     L2
      BKRST   Y1180 K4
      BKRST   Y180 K4
      RST     Y118A
      BKRST   Y1160 K12
1691  LDF     L2
      ORF     X2D
      RST     BL4
      RST     BL3
1697  LDF     X2D
      RST     BL6
1700  LDI     L2
      MOV     K3Y1160 K3Y160
      MOV     K1Y1180 K1Y180
      OUT     T38 K50
      MPS
      LD      Y118A
      ORI     T38
      ANB
      SET     Y18A
      MPP
      ANI     Y118A
      AND     T38
      RST     Y18A
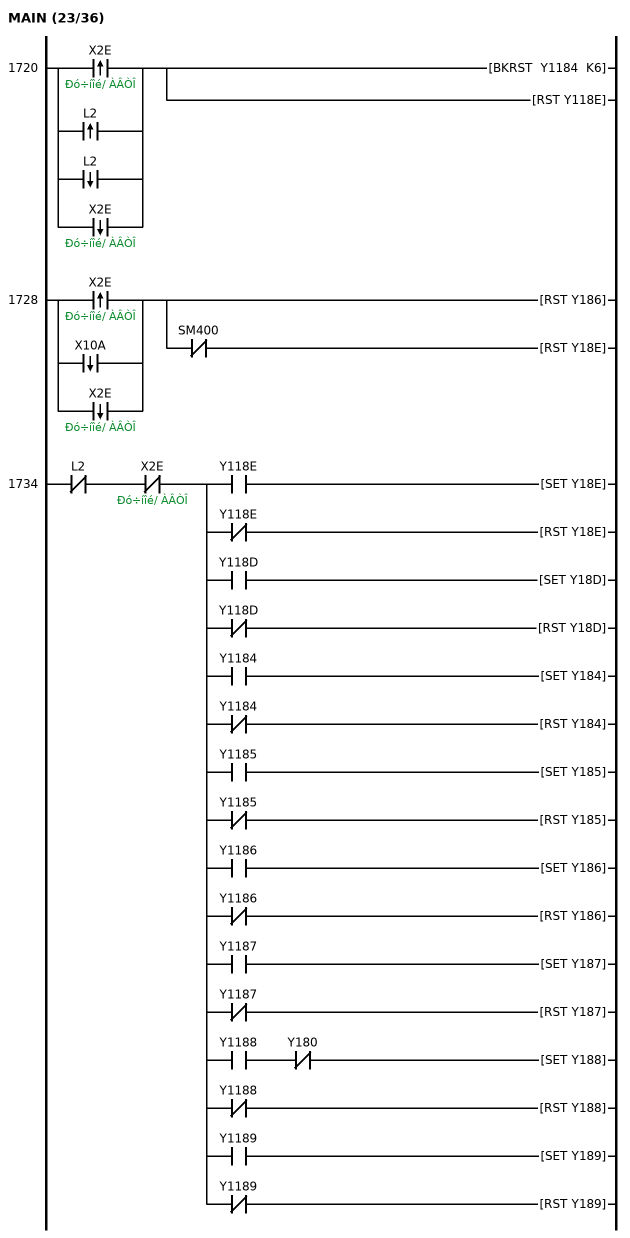
1720  LDP     X2E  ; Ручной/ АВТО
      ORP     L2
      ORF     L2
      ORF     X2E  ; Ручной/ АВТО
      BKRST   Y1184 K6
      RST     Y118E
1728  LDP     X2E  ; Ручной/ АВТО
      ORF     X10A
      ORF     X2E  ; Ручной/ АВТО
      RST     Y186
      ANI     SM400
      RST     Y18E
1734  LDI     L2
      ANI     X2E  ; Ручной/ АВТО
      MPS
      AND     Y118E
      SET     Y18E
      MRD
      ANI     Y118E
      RST     Y18E
      MRD
      AND     Y118D
      SET     Y18D
      MRD
      ANI     Y118D
      RST     Y18D
      MRD
      AND     Y1184
      SET     Y184
      MRD
      ANI     Y1184
      RST     Y184
      MRD
      AND     Y1185
      SET     Y185
      MRD
      ANI     Y1185
      RST     Y185
      MRD
      AND     Y1186
      SET     Y186
      MRD
      ANI     Y1186
      RST     Y186
      MRD
      AND     Y1187
      SET     Y187
      MRD
      ANI     Y1187
      RST     Y187
      MRD
      AND     Y1188
      ANI     Y180
      SET     Y188
      MRD
      ANI     Y1188
      RST     Y188
      MRD
      AND     Y1189
      SET     Y189
      MPP
      ANI     Y1189
      RST     Y189
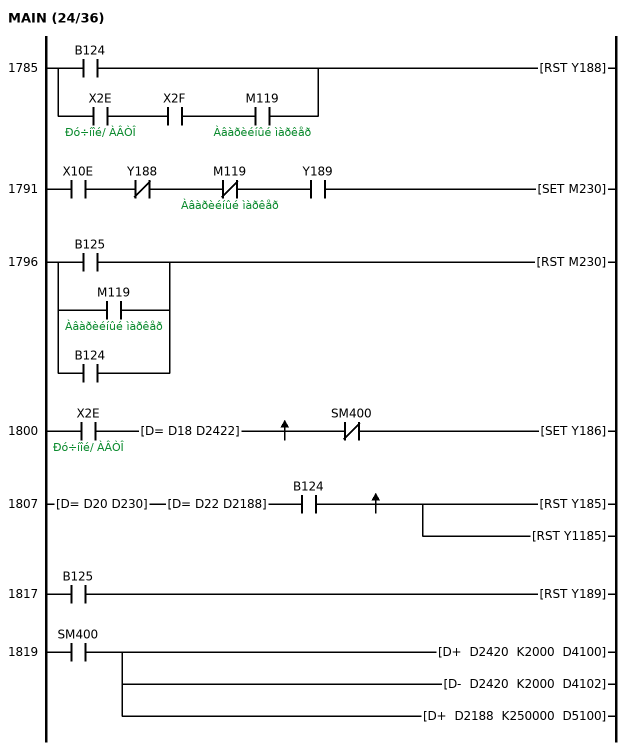
1785  LD      B124
      LD      X2E  ; Ручной/ АВТО
      AND     X2F
      AND     M119  ; Аварийный маркер
      ORB
      RST     Y188
1791  LD      X10E
      ANI     Y188
      ANI     M119  ; Аварийный маркер
      AND     Y189
      SET     M230
1796  LD      B125
      OR      M119  ; Аварийный маркер
      OR      B124
      RST     M230
1800  LD      X2E  ; Ручной/ АВТО
      ANDD=   D18 D2422
      MEP
      ANI     SM400
      SET     Y186
1807  LDD=    D20 D230
      ANDD=   D22 D2188
      AND     B124
      MEP
      RST     Y185
      RST     Y1185
1817  LD      B125
      RST     Y189
1819  LD      SM400
      D+      D2420 K2000 D4100
      D-      D2420 K2000 D4102
      D+      D2188 K250000 D5100
